Xinje XDPPro project, PLC1: XD3-16 (software 3.7.17b 2023-10-13)

PROGRAM Ladder

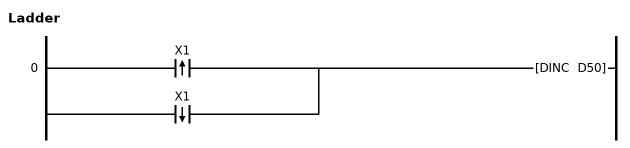
LDP    X1
ORF    X1
DINC   D50